// TIA Portal project "ewon_iolink" (V16)

(* hardware
DEVICE "S7-1200 station_1"  S7-1200 Station
   slot 0: "Rack_0"  S7-1200 Rack  Rack  V1.0
   slot 1: "PLC_1"  CPU 1215C DC/DC/DC  6ES7 215-1AG40-0XB0  V4.4
*)

// ===== PLC "PLC_1"  CPU 1215C DC/DC/DC =====

VAR_GLOBAL   // PLC tag table "Tabla de variables estándar"
   "motor" AT %Q0.0 : Bool;
   "marcha" AT %M810.0 : Bool;
   "paro" AT %M810.1 : Bool;
   "reset" AT %M810.2 : Bool;
   "encendidos" AT %MW813 : Int;
   "motor_var" AT %M816.0 : Bool;
END_VAR

// folder: System blocks/Program resources

DATA_BLOCK "IEC_Counter_0_DB"   // DB2
{ S7_Optimized_Access := 'TRUE' }
AUTHOR : Simatic
FAMILY : IEC
NAME : CNTR
VERSION : 1.0
// stored: InstanceOfName IEC_COUNTER
"IEC_COUNTER"
BEGIN
END_DATA_BLOCK

// folder: (top level)

ORGANIZATION_BLOCK "Main"   // OB1, LAD, ProgramCycle
TITLE = "Main Program Sweep (Cycle)"
{ S7_Optimized_Access := 'TRUE' }
VERSION : 0.1
   VAR_INPUT
      Initial_Call : Bool;   // Initial call of this OB
      Remanence : Bool;   // =True, if remanent data are available
   END_VAR
BEGIN

REGION Network 1
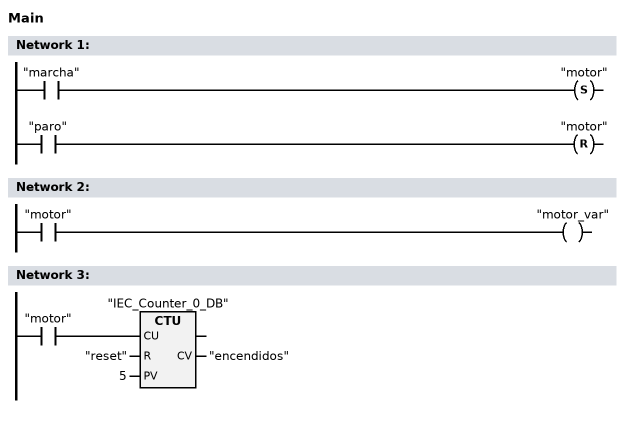
   RUNG wire#powerrail
      Contact( "marcha" )
      S_Coil( "motor" )
   END_RUNG
   RUNG wire#powerrail
      Contact( "paro" )
      R_Coil( "motor" )
   END_RUNG
   // the same network as SCL:
   IF "marcha" THEN "motor" := TRUE; END_IF;
   IF "paro" THEN "motor" := FALSE; END_IF;
END_REGION

REGION Network 2
   RUNG wire#powerrail
      Contact( "motor" )
      Coil( "motor_var" )
   END_RUNG
   // the same network as SCL:
   "motor_var" := "motor";
END_REGION

REGION Network 3
   "IEC_Counter_0_DB".CTU(CU := "motor", R := "reset", PV := 5, CV => "encendidos");
END_REGION
END_ORGANIZATION_BLOCK